// TIA Portal V20 export
VAR_GLOBAL   // PLC tag table "Unit1Em4"
   "BA040AZSBK05.05" AT %I1016.5 : Bool;   // ANODE MAIN P&P1 DETECT SENSOR
   "BA040AZSBK05.06" AT %I1016.6 : Bool;   // ANODE MAIN P&P1 ROTARY CCW
   "BA040AZSBK05.07" AT %I1016.7 : Bool;   // ANODE MAIN P&P1 PRESSURE SWITCH
   "BA040AZSBK05.16" AT %I1017.6 : Bool;   // ANODE MAIN P&P1 ROTARY CW
   "BA040AZSBK06.03" AT %I1020.3 : Bool;   // ANODE MAIN P&P2 DETECT SENSOR
   "BA040AZSBK06.04" AT %I1020.4 : Bool;   // ANODE MAIN P&P2 PRESSURE SWITCH
   "BA040AZSBK09.06" AT %I1032.6 : Bool;   // ANODE ALIGN TABLE ELECTRODE DETECT SENSOR
   "BA040AZSBK09.07" AT %I1032.7 : Bool;   // ANODE ALIGN TABLE PRESSURE SWITCH
   "BA040AZSBK10.00" AT %I1036.0 : Bool;   // ANODE FIX FRONT BACKWARD
   "BA040AZSBK10.02" AT %I1036.2 : Bool;   // ANODE FIX REAR BACKWARD
   "BA040AZSBK10.04" AT %I1036.4 : Bool;   // FIX ANODE DETECT SENSOR
   "BA040AZSBK10.10" AT %I1037.0 : Bool;   // ANODE FIX FRONT FORWARD
   "BA040AZSBK10.12" AT %I1037.2 : Bool;   // ANODE FIX REAR FORWARD
   "BA040AZSBK11.00" AT %I1040.0 : Bool;   // ANODE NG BOX FULL SENSOR
   "BA040AZSBK11.02" AT %I1040.2 : Bool;   // ANODE NG BOX LIFT DOWN
   "BA040AZSBK11.03" AT %I1040.3 : Bool;   // ANODE NG BOX LIFT UP
   "BA040AZSBK11.04" AT %I1040.4 : Bool;   // ANODE NG BOX LOCK DOWN
   "BA040AZSBK11.05" AT %I1040.5 : Bool;   // ANODE NG BOX LOCK UP
   "BA040AZSBK11.06" AT %I1040.6 : Bool;   // ANODE NG BOX NG BOX DETECT SENSOR
   "BA040AZSBK12.00" AT %I1044.0 : Bool;   // ANODE MAIN NG P&P 1st BACKWARD
   "BA040AZSBK12.02" AT %I1044.2 : Bool;   // ANODE MAIN NG P&P 2nd BACKWARD
   "BA040AZSBK12.04" AT %I1044.4 : Bool;   // ANODE MAIN NG P&P UP
   "BA040AZSBK12.06" AT %I1044.6 : Bool;   // ANODE NG P&P VACUUM PRESSURE SWITCH
   "BA040AZSBK12.10" AT %I1045.0 : Bool;   // ANODE MAIN NG P&P 1st FORWARD
   "BA040AZSBK12.12" AT %I1045.2 : Bool;   // ANODE MAIN NG P&P 2nd FORWARD
   "BA040AZSBK12.14" AT %I1045.4 : Bool;   // ANODE MAIN NG P&P DOWN
   "BA040AZSBK12.16" AT %I1045.6 : Bool;   // ANODE NG P&P ELECTRODE DETECT SENSOR
   "BA030AZSSP508.00" AT %I3002.0 : Bool;   // ANODE ALIGN Vision STO // STO - 판정 결과때 같이 살음
   "BA030AZSSP508.01" AT %I3002.1 : Bool;   // ANODE ALIGN VISION JUDGMENT // TRUE = NG, FALSE= OK
   "BA040AZSPM05.00" AT %Q2016.0 : Bool;   // ANODE GLASS CLEANING ON
   "BA040AZSPM05.02" AT %Q2016.2 : Bool;   // ANODE MAIN NG P&P DOWN
   "BA040AZSPM05.03" AT %Q2016.3 : Bool;   // ANODE MAIN NG P&P UP
   "BA040AZSPM05.04" AT %Q2016.4 : Bool;   // ANODE MAIN NG P&P 1st FORWARD
   "BA040AZSPM05.05" AT %Q2016.5 : Bool;   // ANODE MAIN NG P&P 1st BACKWARD
   "BA040AZSPM05.06" AT %Q2016.6 : Bool;   // ANODE MAIN NG P&P 2nd FORWARD
   "BA040AZSPM05.07" AT %Q2016.7 : Bool;   // ANODE MAIN NG P&P 2nd BACKWARD
   "BA040AZSPM05.10" AT %Q2017.0 : Bool;   // ANODE FIX FRONT FORWARD / ANODE FIX REAR FORWARD
   "BA040AZSPM05.11" AT %Q2017.1 : Bool;   // ANODE FIX FRONT BACKWARD / ANODE FIX REAR BACKWARD
   "BA040AZSPM05.12" AT %Q2017.2 : Bool;   // ANODE MAIN P&P#1 Rotary CW
   "BA040AZSPM05.13" AT %Q2017.3 : Bool;   // ANODE MAIN P&P#1 Rotary CCW
   "BA040AZSPM05.14" AT %Q2017.4 : Bool;   // ANODE NG BOX LIFT UP
   "BA040AZSPM05.15" AT %Q2017.5 : Bool;   // ANODE NG BOX LIFT DOWN
   "BA040AZSPM05.16" AT %Q2017.6 : Bool;   // ANODE NG BOX LOCK UP
   "BA040AZSPM05.17" AT %Q2017.7 : Bool;   // ANODE NG BOX LOCK DOWN
   "BA040AZSBK31.00" AT %Q2108.0 : Bool;   // ANODE MAIN P&P#1-1 V/C ON
   "BA040AZSBK31.01" AT %Q2108.1 : Bool;   // ANODE MAIN P&P#1-1 V/C OFF
   "BA040AZSBK31.02" AT %Q2108.2 : Bool;   // ANODE MAIN P&P#2-1 V/C ON
   "BA040AZSBK31.03" AT %Q2108.3 : Bool;   // ANODE MAIN P&P#2-1 V/C OFF
   "BA040AZSBK31.04" AT %Q2108.4 : Bool;   // ANODE MAIN NG P&P V/C ON
   "BA040AZSBK31.05" AT %Q2108.5 : Bool;   // ANODE MAIN NG P&P V/C OFF
   "BA040AZSBK31.06" AT %Q2108.6 : Bool;   // ANODE ALIGN TABLE V/C ON
   "BA040AZSBK31.07" AT %Q2108.7 : Bool;   // ANODE ALIGN TABLE V/C OFF
   "BA040AZSPM01.14" AT %Q2001.4 : Bool;   // ANODE CONVEYOR PICK UP BLOWER ON/OFF
   "BA040AZSPM07.14" AT %Q2025.4 : Bool;   // ANODE CONVEYOR COVER FORWARD
   "BA040AZSPM07.15" AT %Q2025.5 : Bool;   // ANODE CONVEYOR COVER BACKWARD
   "BA040AZSSP504.12" AT %Q3300.2 : Bool;   // ANODE ALIGN VISION CONTROLLER TRIGEER IN
   "BA040AZSBK33.00" AT %Q2208.0 : Bool;   // ANODE MAIN P&P#1-2 V/C ON
   "BA040AZSBK33.01" AT %Q2208.1 : Bool;   // ANODE MAIN P&P#1-2 V/C OFF
   "BA040AZSBK33.04" AT %Q2208.4 : Bool;   // ANODE MAIN P&P#2-2 V/C ON
   "BA040AZSBK33.05" AT %Q2208.5 : Bool;   // ANODE MAIN P&P#2-2 V/C OFF
END_VAR
VAR_GLOBAL CONSTANT   // user constants
   U1EM4_JOB01 : DInt := 1;
   U1EM4_JOB02 : DInt := 2;
   U1EM4_JOB03 : DInt := 3;
   U1EM4_JOB04 : DInt := 4;
   U1EM4_JOB05 : DInt := 5;
   U1EM4_JOB06 : DInt := 6;
   U1EM4_JOB07 : DInt := 7;
   U1EM4_JOB08 : DInt := 8;
   U1EM4_JOB09 : DInt := 9;
   U1EM4_JOB10 : DInt := 10;
   U1EM4_JOB11 : DInt := 11;
   U1EM4_JOB12 : DInt := 12;
   U1EM4_JOB13 : DInt := 13;
   U1EM4_JOB14 : DInt := 14;
   U1EM4_JOB15 : DInt := 15;
   U1EM4_JOB16 : DInt := 16;
   U1EM4_JOB17 : DInt := 17;
   U1EM4_JOB18 : DInt := 18;
   U1EM4_JOB19 : DInt := 19;
   U1EM4_JOB20 : DInt := 20;
   U1EM4_JOB21 : DInt := 21;
   U1EM4_JOB22 : DInt := 22;
   U1EM4_JOB23 : DInt := 23;
   U1EM4_JOB24 : DInt := 24;
   U1EM4_JOB25 : DInt := 25;
   U1EM4_JOB26 : DInt := 26;
   U1EM4_JOB27 : DInt := 27;
   U1EM4_JOB28 : DInt := 28;
   U1EM4_JOB29 : DInt := 29;
   U1EM4_JOB30 : DInt := 30;
   U1EM4_JOB31 : DInt := 31;
   U1EM4_JOB32 : DInt := 32;
   U1EM4_JOB33 : DInt := 33;
   U1EM4_JOB34 : DInt := 34;
   U1EM4_JOB35 : DInt := 35;
   U1EM4_JOB36 : DInt := 36;
   U1EM4_JOB37 : DInt := 37;
   U1EM4_JOB38 : DInt := 38;
   U1EM4_JOB39 : DInt := 39;
   U1EM4_JOB40 : DInt := 40;
   U1EM4_JOB41 : DInt := 41;
   U1EM4_JOB42 : DInt := 42;
   U1EM4_JOB43 : DInt := 43;
   U1EM4_JOB44 : DInt := 44;
   U1EM4_JOB45 : DInt := 45;
   U1EM4_JOB46 : DInt := 46;
   U1EM4_JOB47 : DInt := 47;
   U1EM4_JOB48 : DInt := 48;
   U1EM4_JOB49 : DInt := 49;
   U1EM4_JOB50 : DInt := 50;
   U1EM4_JOB51 : DInt := 51;
   U1EM4_JOB52 : DInt := 52;
   U1EM4_JOB53 : DInt := 53;
   U1EM4_JOB54 : DInt := 54;
   U1EM4_JOB55 : DInt := 55;
   U1EM4_JOB56 : DInt := 56;
   U1EM4_JOB57 : DInt := 57;
   U1EM4_JOB58 : DInt := 58;
   U1EM4_JOB59 : DInt := 59;
   U1EM4_JOB60 : DInt := 60;
   U1EM4_JOB61 : DInt := 61;
   U1EM4_JOB62 : DInt := 62;
   U1EM4_JOB63 : DInt := 63;
   U1EM4_JOB64 : DInt := 64;
   U1EM4_JOB65 : DInt := 65;
   U1EM4_JOB66 : DInt := 66;
   U1EM4_JOB67 : DInt := 67;
   U1EM4_JOB68 : DInt := 68;
   U1EM4_JOB69 : DInt := 69;
   U1EM4_JOB70 : DInt := 70;
   U1EM4_JOB71 : DInt := 71;
   U1EM4_JOB72 : DInt := 72;
   U1EM4_JOB73 : DInt := 73;
   U1EM4_JOB74 : DInt := 74;
   U1EM4_JOB75 : DInt := 75;
   U1EM4_JOB76 : DInt := 76;
   U1EM4_JOB77 : DInt := 77;
   U1EM4_JOB78 : DInt := 78;
   U1EM4_JOB79 : DInt := 79;
   U1EM4_JOB80 : DInt := 80;
   U1EM4_JOB81 : DInt := 81;
   U1EM4_JOB82 : DInt := 82;
   U1EM4_JOB83 : DInt := 83;
   U1EM4_JOB84 : DInt := 84;
   U1EM4_JOB85 : DInt := 85;
   U1EM4_JOB86 : DInt := 86;
   U1EM4_JOB87 : DInt := 87;
   U1EM4_JOB88 : DInt := 88;
   U1EM4_JOB89 : DInt := 89;
   U1EM4_JOB90 : DInt := 90;
   U1EM4_JOB91 : DInt := 91;
   U1EM4_JOB92 : DInt := 92;
   U1EM4_JOB93 : DInt := 93;
   U1EM4_JOB94 : DInt := 94;
   U1EM4_JOB95 : DInt := 95;
   U1EM4_JOB96 : DInt := 96;
   U1EM4_JOB97 : DInt := 97;
   U1EM4_JOB98 : DInt := 98;
   U1EM4_JOB99 : DInt := 99;
   U1EM4_SEQUENCE01 : Int := 1;
   U1EM4_SEQUENCE02 : Int := 2;
   U1EM4_SEQUENCE03 : Int := 3;
   U1EM4_SEQUENCE04 : Int := 4;
   U1EM4_SEQUENCE05 : Int := 5;
   U1EM4_SEQUENCE06 : Int := 6;
   U1EM4_SEQUENCE07 : Int := 7;
   U1EM4_SEQUENCE08 : Int := 8;
   U1EM4_SEQUENCE09 : Int := 9;
   U1EM4_SEQUENCE10 : Int := 10;
   U1EM4_SEQUENCE11 : Int := 11;
   U1EM4_SEQUENCE12 : Int := 12;
   U1EM4_SEQUENCE13 : Int := 13;
   U1EM4_SEQUENCE14 : Int := 14;
   U1EM4_SEQUENCE15 : Int := 15;
   U1EM4_SEQUENCE16 : Int := 16;
   U1EM4_SEQUENCE17 : Int := 17;
   U1EM4_SEQUENCE18 : Int := 18;
   U1EM4_SEQUENCE19 : Int := 19;
   U1EM4_SEQUENCE20 : Int := 20;
   U1EM4_SEQUENCE21 : Int := 21;
   U1EM4_SEQUENCE22 : Int := 22;
   U1EM4_SEQUENCE23 : Int := 23;
   U1EM4_SEQUENCE24 : Int := 24;
   U1EM4_SEQUENCE25 : Int := 25;
   U1EM4_SEQUENCE26 : Int := 26;
   U1EM4_SEQUENCE27 : Int := 27;
   U1EM4_SEQUENCE28 : Int := 28;
   U1EM4_SEQUENCE29 : Int := 29;
   U1EM4_SEQUENCE30 : Int := 30;
   U1EM4_SEQUENCE31 : Int := 31;
   U1EM4_SEQUENCE32 : Int := 32;
   U1EM4_SEQUENCE33 : Int := 33;
   U1EM4_SEQUENCE34 : Int := 34;
   U1EM4_SEQUENCE35 : Int := 35;
   U1EM4_SEQUENCE36 : Int := 36;
   U1EM4_SEQUENCE37 : Int := 37;
   U1EM4_SEQUENCE38 : Int := 38;
   U1EM4_SEQUENCE39 : Int := 39;
   U1EM4_SEQUENCE40 : Int := 40;
   U1EM4_SEQUENCE41 : Int := 41;
   U1EM4_SEQUENCE42 : Int := 42;
   U1EM4_SEQUENCE43 : Int := 43;
   U1EM4_SEQUENCE44 : Int := 44;
   U1EM4_SEQUENCE45 : Int := 45;
   U1EM4_SEQUENCE46 : Int := 46;
   U1EM4_SEQUENCE47 : Int := 47;
   U1EM4_SEQUENCE48 : Int := 48;
   U1EM4_SEQUENCE49 : Int := 49;
   U1EM4_SEQUENCE50 : Int := 50;
   U1EM4_SEQUENCE51 : Int := 51;
   U1EM4_SEQUENCE52 : Int := 52;
   U1EM4_SEQUENCE53 : Int := 53;
   U1EM4_SEQUENCE54 : Int := 54;
   U1EM4_SEQUENCE55 : Int := 55;
   U1EM4_SEQUENCE56 : Int := 56;
   U1EM4_SEQUENCE57 : Int := 57;
   U1EM4_SEQUENCE58 : Int := 58;
   U1EM4_SEQUENCE59 : Int := 59;
   U1EM4_SEQUENCE60 : Int := 60;
   U1EM4_SEQUENCE61 : Int := 61;
   U1EM4_SEQUENCE62 : Int := 62;
   U1EM4_SEQUENCE63 : Int := 63;
   U1EM4_SEQUENCE64 : Int := 64;
   U1EM4_SEQUENCE65 : Int := 65;
   U1EM4_SEQUENCE66 : Int := 66;
   U1EM4_SEQUENCE67 : Int := 67;
   U1EM4_SEQUENCE68 : Int := 68;
   U1EM4_SEQUENCE69 : Int := 69;
   U1EM4_SEQUENCE70 : Int := 70;
   U1EM4_SEQUENCE71 : Int := 71;
   U1EM4_SEQUENCE72 : Int := 72;
   U1EM4_SEQUENCE73 : Int := 73;
   U1EM4_SEQUENCE74 : Int := 74;
   U1EM4_SEQUENCE75 : Int := 75;
   U1EM4_SEQUENCE76 : Int := 76;
   U1EM4_SEQUENCE77 : Int := 77;
   U1EM4_SEQUENCE78 : Int := 78;
   U1EM4_SEQUENCE79 : Int := 79;
   U1EM4_SEQUENCE80 : Int := 80;
   U1EM4_SEQUENCE81 : Int := 81;
   U1EM4_SEQUENCE82 : Int := 82;
   U1EM4_SEQUENCE83 : Int := 83;
   U1EM4_SEQUENCE84 : Int := 84;
   U1EM4_SEQUENCE85 : Int := 85;
   U1EM4_SEQUENCE86 : Int := 86;
   U1EM4_SEQUENCE87 : Int := 87;
   U1EM4_SEQUENCE88 : Int := 88;
   U1EM4_SEQUENCE89 : Int := 89;
   U1EM4_SEQUENCE90 : Int := 90;
   U1EM4_SEQUENCE91 : Int := 91;
   U1EM4_SEQUENCE92 : Int := 92;
   U1EM4_SEQUENCE93 : Int := 93;
   U1EM4_SEQUENCE94 : Int := 94;
   U1EM4_SEQUENCE95 : Int := 95;
   U1EM4_SEQUENCE96 : Int := 96;
   U1EM4_SEQUENCE97 : Int := 97;
   U1EM4_SEQUENCE98 : Int := 98;
   U1EM4_SEQUENCE99 : Int := 99;
   U1EM4_NO_OF_SEQUENCE : USInt := 3;
   U1EM4_NO_OF_AXES : USInt := 8;
   U1EM4_NO_OF_CAM : USInt := 4;
   U1EM4_NO_OF_OUTPUTCAM : USInt := 22;
END_VAR
